FUNCTION_BLOCK FB_RoomTempControl

VAR
	_refHmi			: REFERENCE TO ST_RoomTempHmi;
	_bInit			: BOOL;
	_nCycleTime		: REAL := 0.01;
	_nRoomTemp		: REAL := 20.0;
	_nHeatingRate	: REAL;
	
	// Interfaces
	_iGenerator		: I_Generator;
	
END_VAR


IF _iGenerator.bRunning THEN
	_nHeatingRate := 0.5 * (_iGenerator.nHeat / 100.0) * (_refHmi.nValue / 100.0);
	
	_nRoomTemp := _nRoomTemp + (_nHeatingRate * _nCycleTime);

ELSIF NOT _iGenerator.bRunning THEN
	_nRoomTemp := _nRoomTemp - (0.0005 * _nCycleTime);
	
END_IF

UpdateHmi();

//FB_Init is always available implicitly and it is used primarily for initialization.
//The return value is not evaluated. For a specific influence, you can also declare the
//methods explicitly and provide additional code there with the standard initialization
//code. You can evaluate the return value.
METHOD FB_Init: BOOL
VAR_INPUT
    bInitRetains: BOOL; // TRUE: the retain variables are initialized (reset warm / reset cold)
    bInCopyCode: BOOL;  // TRUE: the instance will be copied to the copy code afterward (online change)   
END_VAR
_bInit := TRUE;
END_METHOD

METHOD Init
VAR_INPUT
	refHmi			: REFERENCE TO ST_RoomTempHmi;
	sName			: STRING;
	iGenerator		: I_Generator;
END_VAR
IF _bInit THEN
	
_refHmi 			REF= refHmi;

_refHmi.sName		:= sName;
_iGenerator			:= iGenerator;

_bInit := FALSE;
END_IF
END_METHOD

METHOD INTERNAL UpdateHmi
VAR_INPUT
END_VAR


_refHmi.nRoomTemperature := _nRoomTemp;
END_METHOD

END_FUNCTION_BLOCK

(* stored: Version 1.1.0.1
   POU FB_RoomTempControl: Id {85271c55-e02b-400b-8b22-1ffc8f0ff4f7}, SpecialFunc None
   Method FB_Init: Id {a8415529-4b20-40d4-b1e3-770eda8edf35}
   Method Init: Id {22fd7ed7-1bd2-4ad5-8128-eea6f8f4e8d2}
   Method UpdateHmi: Id {0c9e6156-ecfc-4699-a54f-b2beaa50eb86} *)
